// TwinCAT 3 PLC project main
// ProgramVersion: 3.1.4024.0
// libraries:
//   Tc2_Standard, * (Beckhoff Automation GmbH)
//   Tc2_System, * (Beckhoff Automation GmbH)
//   Tc3_Module, * (Beckhoff Automation GmbH)
// project tree:
//   / PlcTask.TcTTO
//   POUs/ MAIN.TcPOU
// real-time tasks:
//   TASK PlcTask: cycle T#10ms, priority 20, ADS port 350

CONFIGURATION main
    RESOURCE PLC ON TwinCAT3
        TASK PlcTask(INTERVAL := T#10ms, PRIORITY := 20);
        PROGRAM MAIN WITH PlcTask : MAIN;
    END_RESOURCE
END_CONFIGURATION

// ---- POUs/MAIN.TcPOU
PROGRAM MAIN
VAR
	bS1 : INT; //Sensor 1
	bS2 : INT; //Sensor 2
	bS3 : INT; //Sensor 3
	
	bL1 : BOOL; //Lamp 1
	bL2 : BOOL; //Lamp 2
	bL3 : BOOL; //Lamp 3
	bL4 : BOOL; //Lamp 4
	bL5 : BOOL; //Lamp 5
	
END_VAR

//We herhalen de oefening van de alarmbewaking. We maken nu echter gebruik van simpele analoge sensoren.
//We moeten nu de drempelwaarden die we normaal in onze smart sensor zouden ingesteld hebben aan het programma moeten meegeven.
//Deze zijn voor de druk, temperatuur en vloeistofniveau respectievelijk 12, 80 en 22.
//Het programma dat we geschreven hebben voor onze 5 lampen blijft zo goed als hetzelfde.

bL1 := INT_TO_BOOL(bS1 > 12);
bL2 := INT_TO_BOOL(bS2 > 80);
bL3 := int_to_bool(bS3 > 22);

END_PROGRAM
